# EPICS autosave request: GalilSup/Db/galil_analog_in.req
$(P)$(R)_MON.DESC
$(P)$(R)Deadb_SP.VAL
